{attribute 'qualified_only'}
VAR_GLOBAL CONSTANT
	nBufferLength:			UINT:= 100;
	nHmiLength:				UINT:= 50;
END_VAR

(* stored: Version 1.1.0.1
   GVL Parameters: Id {8015e61c-8c09-4deb-9bf8-f40387a603ee}, ParameterList True *)
